TYPE ST_AxisCtrlV2 :
STRUCT
    Io                        :ST_AxisIo;  (*轴IO信号*)
    Status                  :ST_AxisStatus;  
    Cmd                    :ST_AxisCmdV2;  
END_STRUCT
END_TYPE

(* stored: Version 1.1.0.1, ProductVersion 3.1.4024.9
   DUT ST_AxisCtrlV2: Id {ec255e07-db00-4c2a-8447-6d137b95e3ee} *)
